Yaskawa INFORM job: EARCUT.JBI

/JOB
//NAME EARCUT
//POS
///NPOS 14,0,0,0,0,0
///TOOL 0
///POSTYPE PULSE
///PULSE
C00000=-238997,-175100,-128752,-104159,-111414,-73968
C00001=-71507,-161626,-119118,-161080,-39585,7669
C00002=-82126,-163457,-110199,-154374,-34145,678
C00003=-79523,-164634,-107653,-154379,-31740,1281
C00004=-115197,-167761,-107678,-141941,-42334,-16259
C00005=-160791,-167181,-107379,-141930,-59879,-31286
C00006=-176784,-164790,-110014,-144695,-67811,-35093
C00007=-173984,-163323,-108663,-144323,-66852,-34231
C00008=-192692,-162241,-113776,-147886,-76073,-38816
C00009=-203913,-155132,-116176,-150470,-84008,-40866
C00010=-210193,-148688,-117230,-151858,-89420,-41838
C00011=-211379,-145644,-116893,-152105,-91033,-41858
C00012=-214137,-139010,-117103,-152597,-95031,-41854
C00013=-215967,-147507,-131505,-151076,-96597,-41897
//INST
///DATE 2023/09/18 18:33
///ATTR SC,RW
///GROUP1 RB1
NOP
MOVJ C00000 VJ=12.50
MOVJ C00001 VJ=12.50
MOVJ C00002 VJ=12.50
COMM MOVJ C00003 VJ=12.50
MOVS C00004 V=16.0
COMM MOVS C00005 V=16.0
COMM MOVS C00006 V=16.0
MOVS C00007 V=16.0
COMM MOVS C00008 V=16.0
COMM MOVS C00009 V=16.0
COMM MOVS C00010 V=16.0
COMM MOVS C00011 V=16.0
MOVS C00012 V=16.0
MOVL C00013 V=200.0
END
